// Mitsubishi GX Works2 project: PLC_master   PLC: Q06UDV
// program mas Indra

PROGRAM MAIN
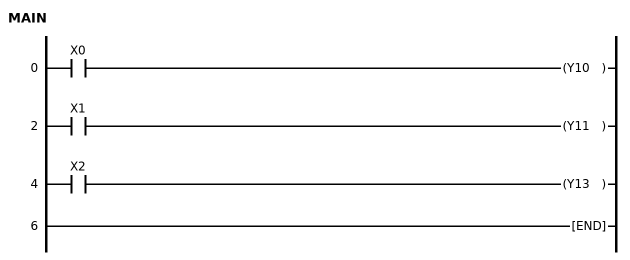
0     LD      X0
      OUT     Y10
2     LD      X1
      OUT     Y11
4     LD      X2
      OUT     Y13
6     END
END_PROGRAM

PROGRAM PCB
0     END
END_PROGRAM
